ABB RobotStudio station: Lab1.11.rsstn

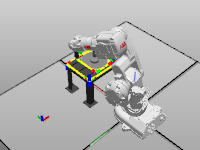
Station Lab1.10 (saved by RobotStudio 21.2.9526.0)
Controller IRB140_6_81
  mechanical unit ROB_1: IRB140_6_81_C_03, 6 joints, base frame (0, 0, 0) mm
Layout (positions relative to the parent item):
  - IRB140_6_81_C_03 [mechanism, from Robots\IRB140_6_81_C_G_03.rslib] at (0, 0, 0) mm; joint values [0.1651, 0.5626, -0.138, 0, 1.1463, -1.4056] (rad or m)
  - UISpenholder [mechanism, from RS1\UISpenholder.rslib] at (600, 100, 435) mm, rotated rx -180 ry 0 rz -90 deg
  - table_and_fixture_140 [part, from Training Objects\propeller_table.rslib] at (300, 225, 0) mm, rotated rx 0 ry 0 rz -90 deg
Attachment: UISpenholder is attached to IRB140_6_81_C_03 / Link6
Attachment: WobjTable is attached to table_and_fixture_140
Collision set CollisionSet_1: UISpenholder against table_and_fixture_140, near miss 0 m
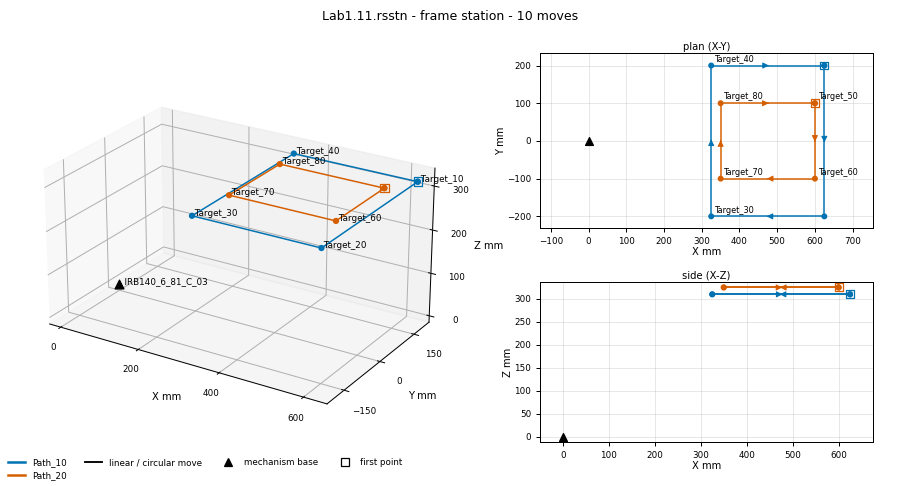
[picture p0: tool path of Lab1.11.rsstn in frame station, 10 of 10 moves have a stored position in this frame; points joined in program order, loops and branches not executed]
Targets, tools, work objects and paths stored in the station, written as RAPID:
! task T_ROB1
MODULE Module1
  PERS tooldata UISpenholder:=[TRUE,[[0,0,110],[1,0,0,0]],[1,[0,0,1],[1,0,0,0],0,0,0]];
  TASK PERS wobjdata WobjTable:=[FALSE,TRUE,"",[[475,625,2],[0.707106781,0,0,-0.707106781]],[[425,-150,308],[1,0,0,0]]];
  CONST robtarget Target_10:=[[0,300,0],[0,1,0,0],[0,0,0,0],[9E+09,9E+09,9E+09,9E+09,9E+09,9E+09]];
  CONST robtarget Target_20:=[[400,300,0],[0,-0.707106781,0.707106781,0],[-1,0,-1,0],[9E+09,9E+09,9E+09,9E+09,9E+09,9E+09]];
  CONST robtarget Target_30:=[[400,0,0],[0,0,1,0],[-1,0,0,0],[9E+09,9E+09,9E+09,9E+09,9E+09,9E+09]];
  CONST robtarget Target_40:=[[0,0,0],[0,0.707106781,0.707106781,0],[0,0,-2,0],[9E+09,9E+09,9E+09,9E+09,9E+09,9E+09]];
  CONST robtarget Target_50:=[[100,275,15],[0,1,0,0],[0,0,0,0],[9E+09,9E+09,9E+09,9E+09,9E+09,9E+09]];
  CONST robtarget Target_60:=[[300,275,15],[0,-0.707106781,0.707106781,0],[-1,0,-1,0],[9E+09,9E+09,9E+09,9E+09,9E+09,9E+09]];
  CONST robtarget Target_70:=[[300,25,15],[0,0,1,0],[-1,0,0,0],[9E+09,9E+09,9E+09,9E+09,9E+09,9E+09]];
  CONST robtarget Target_80:=[[100,25,15],[0,0.707106781,0.707106781,0],[0,0,-2,0],[9E+09,9E+09,9E+09,9E+09,9E+09,9E+09]];
  PROC Path_10()
    MoveL Target_10,v1000,z5,UISpenholder\WObj:=WobjTable;
    MoveL Target_20,v1000,z5,UISpenholder\WObj:=WobjTable;
    MoveL Target_30,v1000,z5,UISpenholder\WObj:=WobjTable;
    MoveL Target_40,v1000,z5,UISpenholder\WObj:=WobjTable;
    MoveL Target_10,v1000,z5,UISpenholder\WObj:=WobjTable;
  ENDPROC
  PROC Path_20()
    MoveL Target_50,v1000,z100,UISpenholder\WObj:=WobjTable;
    MoveL Target_60,v1000,z100,UISpenholder\WObj:=WobjTable;
    MoveL Target_70,v1000,z100,UISpenholder\WObj:=WobjTable;
    MoveL Target_80,v1000,z100,UISpenholder\WObj:=WobjTable;
    MoveL Target_50,v1000,z100,UISpenholder\WObj:=WobjTable;
  ENDPROC
ENDMODULE

